FUNCTION_BLOCK FB_FakeAxis_BaseUnit EXTENDS FB_BaseUnit IMPLEMENTS I_Axis_BaseUnit
VAR
	_bAxisIsDisabled : BOOL;
	_bAxisHasJob : BOOL;
	_fAxisActualPosition : LREAL;
	_fAxisActualVelocity : LREAL;
	_nCycle : UDINT;
	_nCallSequence : UDINT;

	_aScripts : ARRAY[1..32] OF ST_FakeAxisScriptStep;
	_nScriptCount : UINT;
	_bScriptOverflowed : BOOL;
	_bScriptConfigurationError : BOOL;

	_aHistory : ARRAY[1..256] OF ST_FakeAxisCall;
	_nHistoryCount : UINT;
	_bHistoryOverflowed : BOOL;

	_bJogActive : BOOL;
	_bMoveAbsActive : BOOL;
	_bMoveVelActive : BOOL;
	_bStopActive : BOOL;
	_bResetActive : BOOL;
	_bHaltActive : BOOL;

	_bJogDone : BOOL;
	_bJogInVelocity : BOOL;
	_bJogError : BOOL;
	_nJogErrorId : UDINT;
	_bMoveAbsDone : BOOL;
	_bMoveAbsInVelocity : BOOL;
	_bMoveAbsError : BOOL;
	_nMoveAbsErrorId : UDINT;
	_bMoveVelDone : BOOL;
	_bMoveVelInVelocity : BOOL;
	_bMoveVelError : BOOL;
	_nMoveVelErrorId : UDINT;
	_bStopDone : BOOL;
	_bStopInVelocity : BOOL;
	_bStopError : BOOL;
	_nStopErrorId : UDINT;
	_bResetDone : BOOL;
	_bResetInVelocity : BOOL;
	_bResetError : BOOL;
	_nResetErrorId : UDINT;
	_bHaltDone : BOOL;
	_bHaltInVelocity : BOOL;
	_bHaltError : BOOL;
	_nHaltErrorId : UDINT;
END_VAR

M_CyclicUpdate();

PROPERTY AxisActualPosition : LREAL
GET
AxisActualPosition := _fAxisActualPosition;
END_GET
END_PROPERTY

PROPERTY AxisActualVelocity : LREAL
GET
AxisActualVelocity := _fAxisActualVelocity;
END_GET
END_PROPERTY

PROPERTY AxisHasJob : BOOL
GET
AxisHasJob := _bAxisHasJob;
END_GET
END_PROPERTY

PROPERTY AxisIsDisabled : BOOL
GET
AxisIsDisabled := _bAxisIsDisabled;
END_GET
END_PROPERTY

PROPERTY CurrentCycle : UDINT
GET
CurrentCycle := _nCycle;
END_GET
END_PROPERTY

PROPERTY HistoryCount : UINT
GET
HistoryCount := _nHistoryCount;
END_GET
END_PROPERTY

PROPERTY HistoryOverflowed : BOOL
GET
HistoryOverflowed := _bHistoryOverflowed;
END_GET
END_PROPERTY

METHOD M_ClearCallHistory
VAR_INPUT
END_VAR
MEMSET(ADR(_aHistory), 0, SIZEOF(_aHistory));
_nHistoryCount := 0;
_nCallSequence := 0;
_bHistoryOverflowed := FALSE;
END_METHOD

METHOD M_CyclicUpdate
VAR_INPUT
END_VAR
_nCycle := _nCycle + 1;

M_ProcessOperation(
	Operation := E_FakeAxisOperation.Jog,
	Active := _bJogActive,
	Done := _bJogDone,
	InVelocity := _bJogInVelocity,
	Error := _bJogError,
	ErrorId := _nJogErrorId
);
M_ProcessOperation(
	Operation := E_FakeAxisOperation.MoveAbs,
	Active := _bMoveAbsActive,
	Done := _bMoveAbsDone,
	InVelocity := _bMoveAbsInVelocity,
	Error := _bMoveAbsError,
	ErrorId := _nMoveAbsErrorId
);
M_ProcessOperation(
	Operation := E_FakeAxisOperation.MoveVel,
	Active := _bMoveVelActive,
	Done := _bMoveVelDone,
	InVelocity := _bMoveVelInVelocity,
	Error := _bMoveVelError,
	ErrorId := _nMoveVelErrorId
);
M_ProcessOperation(
	Operation := E_FakeAxisOperation.Stop,
	Active := _bStopActive,
	Done := _bStopDone,
	InVelocity := _bStopInVelocity,
	Error := _bStopError,
	ErrorId := _nStopErrorId
);
M_ProcessOperation(
	Operation := E_FakeAxisOperation.Reset,
	Active := _bResetActive,
	Done := _bResetDone,
	InVelocity := _bResetInVelocity,
	Error := _bResetError,
	ErrorId := _nResetErrorId
);
M_ProcessOperation(
	Operation := E_FakeAxisOperation.Halt,
	Active := _bHaltActive,
	Done := _bHaltDone,
	InVelocity := _bHaltInVelocity,
	Error := _bHaltError,
	ErrorId := _nHaltErrorId
);
END_METHOD

METHOD M_GetCall : BOOL
VAR_INPUT
	Index : UINT;
END_VAR
VAR_OUTPUT
	CallRecord : ST_FakeAxisCall;
END_VAR
M_GetCall := FALSE;
MEMSET(ADR(CallRecord), 0, SIZEOF(CallRecord));
IF (Index = 0) OR (Index > _nHistoryCount) THEN
	RETURN;
END_IF
CallRecord := _aHistory[Index];
M_GetCall := TRUE;
END_METHOD

METHOD M_Halt : BOOL
VAR_INPUT
	OwnerId : T_ResourceOwnerId;
	Execute : BOOL;
	Deceleration : LREAL;
END_VAR
VAR_OUTPUT
	Done : BOOL;
	Error : BOOL;
END_VAR
VAR
	bAccepted : BOOL;
END_VAR
bAccepted := M_IsResourceOwner(OwnerId := OwnerId);
M_RecordCall(
	Operation := E_FakeAxisOperation.Halt,
	OwnerId := OwnerId,
	Accepted := bAccepted,
	Execute := Execute,
	JogForward := FALSE,
	JogBackwards := FALSE,
	Mode := E_JogMode.MC_JOGMODE_CONTINOUS,
	Direction := MC_Direction.MC_Positive_Direction,
	Position := 0,
	Velocity := 0,
	Acceleration := 0,
	Deceleration := Deceleration
);

M_Halt := bAccepted;
IF NOT bAccepted THEN
	Done := FALSE;
	Error := FALSE;
	RETURN;
END_IF

_bHaltActive := Execute;
Done := _bHaltDone;
Error := _bHaltError;
END_METHOD

METHOD M_Jog : BOOL
VAR_INPUT
	OwnerId : T_ResourceOwnerId;
	JogForward : BOOL;
	JogBackwards : BOOL;
	Mode : E_JogMode;
	Position : LREAL;
	Velocity : LREAL;
	Acceleration : LREAL;
	Deceleration : LREAL;
END_VAR
VAR_OUTPUT
	Done : BOOL;
	Error : BOOL;
	ErrorId : UDINT;
END_VAR
VAR
	bAccepted : BOOL;
END_VAR
bAccepted := M_IsResourceOwner(OwnerId := OwnerId);
M_RecordCall(
	Operation := E_FakeAxisOperation.Jog,
	OwnerId := OwnerId,
	Accepted := bAccepted,
	Execute := JogForward OR JogBackwards,
	JogForward := JogForward,
	JogBackwards := JogBackwards,
	Mode := Mode,
	Direction := MC_Direction.MC_Positive_Direction,
	Position := Position,
	Velocity := Velocity,
	Acceleration := Acceleration,
	Deceleration := Deceleration
);

M_Jog := bAccepted;
IF NOT bAccepted THEN
	Done := FALSE;
	Error := FALSE;
	ErrorId := 0;
	RETURN;
END_IF

_bJogActive := JogForward OR JogBackwards;
Done := _bJogDone;
Error := _bJogError;
ErrorId := _nJogErrorId;
END_METHOD

METHOD M_MoveAbs : BOOL
VAR_INPUT
	OwnerId : T_ResourceOwnerId;
	Execute : BOOL;
	Position : LREAL;
	Velocity : LREAL;
	Acceleration : LREAL;
	Deceleration : LREAL;
END_VAR
VAR_OUTPUT
	Done : BOOL;
	Error : BOOL;
	ErrorId : UDINT;
END_VAR
VAR
	bAccepted : BOOL;
END_VAR
bAccepted := M_IsResourceOwner(OwnerId := OwnerId);
M_RecordCall(
	Operation := E_FakeAxisOperation.MoveAbs,
	OwnerId := OwnerId,
	Accepted := bAccepted,
	Execute := Execute,
	JogForward := FALSE,
	JogBackwards := FALSE,
	Mode := E_JogMode.MC_JOGMODE_CONTINOUS,
	Direction := MC_Direction.MC_Positive_Direction,
	Position := Position,
	Velocity := Velocity,
	Acceleration := Acceleration,
	Deceleration := Deceleration
);

M_MoveAbs := bAccepted;
IF NOT bAccepted THEN
	Done := FALSE;
	Error := FALSE;
	ErrorId := 0;
	RETURN;
END_IF

_bMoveAbsActive := Execute;
Done := _bMoveAbsDone;
Error := _bMoveAbsError;
ErrorId := _nMoveAbsErrorId;
END_METHOD

METHOD M_MoveVel : BOOL
VAR_INPUT
	OwnerId : T_ResourceOwnerId;
	Execute : BOOL;
	Direction : MC_Direction;
	Velocity : LREAL;
	Acceleration : LREAL;
	Deceleration : LREAL;
END_VAR
VAR_OUTPUT
	InVelocity : BOOL;
	Error : BOOL;
END_VAR
VAR
	bAccepted : BOOL;
END_VAR
bAccepted := M_IsResourceOwner(OwnerId := OwnerId);
M_RecordCall(
	Operation := E_FakeAxisOperation.MoveVel,
	OwnerId := OwnerId,
	Accepted := bAccepted,
	Execute := Execute,
	JogForward := FALSE,
	JogBackwards := FALSE,
	Mode := E_JogMode.MC_JOGMODE_CONTINOUS,
	Direction := Direction,
	Position := 0,
	Velocity := Velocity,
	Acceleration := Acceleration,
	Deceleration := Deceleration
);

M_MoveVel := bAccepted;
IF NOT bAccepted THEN
	InVelocity := FALSE;
	Error := FALSE;
	RETURN;
END_IF

_bMoveVelActive := Execute;
InVelocity := _bMoveVelInVelocity;
Error := _bMoveVelError;
END_METHOD

METHOD PRIVATE M_ProcessOperation
VAR_INPUT
	Operation : E_FakeAxisOperation;
	Active : BOOL;
END_VAR
VAR_IN_OUT
	Done : BOOL;
	InVelocity : BOOL;
	Error : BOOL;
	ErrorId : UDINT;
END_VAR
VAR
	nIndex : UINT;
END_VAR
Done := FALSE;
InVelocity := FALSE;
Error := FALSE;
ErrorId := 0;

FOR nIndex := 1 TO _nScriptCount DO
	IF (_aScripts[nIndex].Operation = Operation) AND NOT _aScripts[nIndex].Consumed THEN

		// Label script that is consumed
		IF NOT Active THEN
			IF _aScripts[nIndex].Started THEN
				_aScripts[nIndex].Consumed := TRUE;
			END_IF
			RETURN;
		END_IF

		// Start managing script
		IF NOT _aScripts[nIndex].Started THEN
			_aScripts[nIndex].Started := TRUE;
			_aScripts[nIndex].ActiveCycles := 0;
		END_IF

		// Manage AfterActiveCycle
		IF NOT _aScripts[nIndex].ResultLatched THEN
			_aScripts[nIndex].ActiveCycles := _aScripts[nIndex].ActiveCycles + 1;
			IF (_aScripts[nIndex].AfterActiveCycles = 0)
				OR (_aScripts[nIndex].ActiveCycles >= _aScripts[nIndex].AfterActiveCycles) THEN
			_aScripts[nIndex].ResultLatched := TRUE;
		END_IF
	END_IF

	// Output result if after certain active cycles
	IF _aScripts[nIndex].ResultLatched THEN
		Done := _aScripts[nIndex].Done;
		InVelocity := _aScripts[nIndex].InVelocity;
		Error := _aScripts[nIndex].Error;
		ErrorId := _aScripts[nIndex].ErrorId;
	END_IF
	RETURN;
END_IF
END_FOR
END_METHOD

METHOD M_QueueResult : BOOL
VAR_INPUT
	Operation : E_FakeAxisOperation;
	AfterActiveCycles : UINT;
	Done : BOOL;
	InVelocity : BOOL;
	Error : BOOL;
	ErrorId : UDINT;
END_VAR
M_QueueResult := FALSE;

IF (Operation = E_FakeAxisOperation.None) OR (Done AND Error) THEN
	_bScriptConfigurationError := TRUE;
	RETURN;
END_IF

IF _nScriptCount >= 32 THEN
	_bScriptOverflowed := TRUE;
	RETURN;
END_IF

_nScriptCount := _nScriptCount + 1;
_aScripts[_nScriptCount].Operation := Operation;
_aScripts[_nScriptCount].AfterActiveCycles := AfterActiveCycles;
_aScripts[_nScriptCount].Done := Done;
_aScripts[_nScriptCount].InVelocity := InVelocity;
_aScripts[_nScriptCount].Error := Error;
_aScripts[_nScriptCount].ErrorId := ErrorId;
M_QueueResult := TRUE;
END_METHOD

METHOD PRIVATE M_RecordCall
VAR_INPUT
	Operation : E_FakeAxisOperation;
	OwnerId : T_ResourceOwnerId;
	Accepted : BOOL;
	Execute : BOOL;
	JogForward : BOOL;
	JogBackwards : BOOL;
	Mode : E_JogMode;
	Direction : MC_Direction;
	Position : LREAL;
	Velocity : LREAL;
	Acceleration : LREAL;
	Deceleration : LREAL;
END_VAR
_nCallSequence := _nCallSequence + 1;
IF _nHistoryCount >= 256 THEN
	_bHistoryOverflowed := TRUE;
	RETURN;
END_IF

_nHistoryCount := _nHistoryCount + 1;
_aHistory[_nHistoryCount].Sequence := _nCallSequence;
_aHistory[_nHistoryCount].Cycle := _nCycle;
_aHistory[_nHistoryCount].Operation := Operation;
_aHistory[_nHistoryCount].OwnerId := OwnerId;
_aHistory[_nHistoryCount].Accepted := Accepted;
_aHistory[_nHistoryCount].Execute := Execute;
_aHistory[_nHistoryCount].JogForward := JogForward;
_aHistory[_nHistoryCount].JogBackwards := JogBackwards;
_aHistory[_nHistoryCount].Mode := Mode;
_aHistory[_nHistoryCount].Direction := Direction;
_aHistory[_nHistoryCount].Position := Position;
_aHistory[_nHistoryCount].Velocity := Velocity;
_aHistory[_nHistoryCount].Acceleration := Acceleration;
_aHistory[_nHistoryCount].Deceleration := Deceleration;
END_METHOD

METHOD M_Reset : BOOL
VAR_INPUT
	OwnerId : T_ResourceOwnerId;
	Execute : BOOL;
END_VAR
VAR_OUTPUT
	Done : BOOL;
	Error : BOOL;
	ErrorId : UDINT;
END_VAR
VAR
	bAccepted : BOOL;
END_VAR
bAccepted := M_IsResourceOwner(OwnerId := OwnerId);
M_RecordCall(
	Operation := E_FakeAxisOperation.Reset,
	OwnerId := OwnerId,
	Accepted := bAccepted,
	Execute := Execute,
	JogForward := FALSE,
	JogBackwards := FALSE,
	Mode := E_JogMode.MC_JOGMODE_CONTINOUS,
	Direction := MC_Direction.MC_Positive_Direction,
	Position := 0,
	Velocity := 0,
	Acceleration := 0,
	Deceleration := 0
);

M_Reset := bAccepted;
IF NOT bAccepted THEN
	Done := FALSE;
	Error := FALSE;
	ErrorId := 0;
	RETURN;
END_IF

_bResetActive := Execute;
Done := _bResetDone;
Error := _bResetError;
ErrorId := _nResetErrorId;
END_METHOD

METHOD M_ResetScenario
VAR_INPUT
END_VAR
_ResourceOwnerId := 0;
_bAxisIsDisabled := FALSE;
_bAxisHasJob := FALSE;
_fAxisActualPosition := 0;
_fAxisActualVelocity := 0;
_nCycle := 0;
_nScriptCount := 0;
_bScriptOverflowed := FALSE;
_bScriptConfigurationError := FALSE;
MEMSET(ADR(_aScripts), 0, SIZEOF(_aScripts));
M_ClearCallHistory();

_bJogActive := FALSE;
_bMoveAbsActive := FALSE;
_bMoveVelActive := FALSE;
_bStopActive := FALSE;
_bResetActive := FALSE;
_bHaltActive := FALSE;
_bJogDone := FALSE;
_bJogInVelocity := FALSE;
_bJogError := FALSE;
_nJogErrorId := 0;
_bMoveAbsDone := FALSE;
_bMoveAbsInVelocity := FALSE;
_bMoveAbsError := FALSE;
_nMoveAbsErrorId := 0;
_bMoveVelDone := FALSE;
_bMoveVelInVelocity := FALSE;
_bMoveVelError := FALSE;
_nMoveVelErrorId := 0;
_bStopDone := FALSE;
_bStopInVelocity := FALSE;
_bStopError := FALSE;
_nStopErrorId := 0;
_bResetDone := FALSE;
_bResetInVelocity := FALSE;
_bResetError := FALSE;
_nResetErrorId := 0;
_bHaltDone := FALSE;
_bHaltInVelocity := FALSE;
_bHaltError := FALSE;
_nHaltErrorId := 0;
END_METHOD

METHOD M_SetAxisFeedback
VAR_INPUT
	ActualPosition : LREAL;
	ActualVelocity : LREAL;
END_VAR
_fAxisActualPosition := ActualPosition;
_fAxisActualVelocity := ActualVelocity;
END_METHOD

METHOD M_SetAxisState
VAR_INPUT
	Disabled : BOOL;
	HasJob : BOOL;
END_VAR
_bAxisIsDisabled := Disabled;
_bAxisHasJob := HasJob;
END_METHOD

METHOD M_Stop : BOOL
VAR_INPUT
	OwnerId : T_ResourceOwnerId;
	Execute : BOOL;
	Deceleration : LREAL;
END_VAR
VAR_OUTPUT
	Done : BOOL;
	Error : BOOL;
	ErrorId : UDINT;
END_VAR
VAR
	bAccepted : BOOL;
END_VAR
bAccepted := M_IsResourceOwner(OwnerId := OwnerId);
M_RecordCall(
	Operation := E_FakeAxisOperation.Stop,
	OwnerId := OwnerId,
	Accepted := bAccepted,
	Execute := Execute,
	JogForward := FALSE,
	JogBackwards := FALSE,
	Mode := E_JogMode.MC_JOGMODE_CONTINOUS,
	Direction := MC_Direction.MC_Positive_Direction,
	Position := 0,
	Velocity := 0,
	Acceleration := 0,
	Deceleration := Deceleration
);

M_Stop := bAccepted;
IF NOT bAccepted THEN
	Done := FALSE;
	Error := FALSE;
	ErrorId := 0;
	RETURN;
END_IF

_bStopActive := Execute;
Done := _bStopDone;
Error := _bStopError;
ErrorId := _nStopErrorId;
END_METHOD

PROPERTY ScriptConfigurationError : BOOL
GET
ScriptConfigurationError := _bScriptConfigurationError;
END_GET
END_PROPERTY

PROPERTY ScriptOverflowed : BOOL
GET
ScriptOverflowed := _bScriptOverflowed;
END_GET
END_PROPERTY

END_FUNCTION_BLOCK

(* stored: Version 1.1.0.1, ProductVersion 3.1.4026.18
   POU FB_FakeAxis_BaseUnit: Id {e3e8b765-2c8e-48cb-88c1-18c6481deefe}, SpecialFunc None
   Property AxisActualPosition: Id {c803e875-2d0d-4296-9bc7-ab55d60b4a28}
   Get Get: Id {bb61b1fe-e7db-4677-a8e6-bd4dbf4da4e1}
   Property AxisActualVelocity: Id {78b99b62-4a3f-4ce6-bd76-f215a6374ec7}
   Get Get: Id {627ebdf8-75c0-44ee-8666-e67c59e60c18}
   Property AxisHasJob: Id {28149424-d35b-4967-a2b8-84de1d190c02}
   Get Get: Id {d07beebe-b038-4ceb-8984-0b7cdced23b2}
   Property AxisIsDisabled: Id {0319dfcd-7dbc-4acf-a420-3b38d7710e27}
   Get Get: Id {980df56c-f78c-4645-a521-29c7cb19d811}
   Property CurrentCycle: Id {41621bfd-1eb9-4fd5-a0a4-82ffea373ca6}
   Get Get: Id {724f2233-06dd-4319-8477-e87fb17fa22d}
   Property HistoryCount: Id {3fb77f6b-f796-4033-81b5-f81aca9a5cce}
   Get Get: Id {a50cdb82-650a-4b79-9503-ce96d9a01cb3}
   Property HistoryOverflowed: Id {43c86ec2-a45e-4a9a-818f-6de5e3f937c7}
   Get Get: Id {6a144965-58c8-45ce-857b-8e1b1074555f}
   Method M_ClearCallHistory: Id {f089176f-389b-4baa-a2da-4f354ec5d7f3}
   Method M_CyclicUpdate: Id {51353dc4-27da-4cdc-9e93-0412f19d6e2c}
   Method M_GetCall: Id {94ad7b50-f13b-43b4-a754-adcb1517e88f}
   Method M_Halt: Id {6eead5a4-5f3f-43d9-aa96-68d42a79be0a}
   Method M_Jog: Id {5e662ea3-bf75-47da-a7ed-fc6bb775a22a}
   Method M_MoveAbs: Id {799e5942-56df-4f9f-b9ff-c946088a2daf}
   Method M_MoveVel: Id {0cc6eabc-5d4d-4943-826e-9307a0401b16}
   Method M_ProcessOperation: Id {1ccb0dd7-a7b9-4452-8393-44608ab6d1e1}
   Method M_QueueResult: Id {b0f97812-5ba5-4585-b056-83a9174ddfb3}
   Method M_RecordCall: Id {46ae4ea2-55f9-42d6-af9b-1610838d9b64}
   Method M_Reset: Id {1a644686-8406-49fb-9498-3fde4ac973cb}
   Method M_ResetScenario: Id {de0840d9-c339-43cb-8bf8-ae01686058c7}
   Method M_SetAxisFeedback: Id {82b4c35c-c729-464f-b941-dd0e760a7934}
   Method M_SetAxisState: Id {10c2eb70-a53b-4b94-8710-7bc4d3c0b6f3}
   Method M_Stop: Id {51ed3baa-d27d-4af9-9931-fc510a406353}
   Property ScriptConfigurationError: Id {6c11b652-02b9-4680-a22d-45f650b44c03}
   Get Get: Id {2082a054-a11a-4812-aab3-726089b22a5c}
   Property ScriptOverflowed: Id {0aa8b35c-6e9b-42d4-9127-9edbc51faebe}
   Get Get: Id {2e632f4c-7e78-46e5-91f0-8619a0fa4555} *)
